FUNCTION MeasureUnits_to_Count : int;
VAR_INPUT
	iValue_in	: INT; 
	iHigh		: REAL;
	iLow		: REAL;
END_VAR
VAR
END_VAR

MeasureUnits_to_Count	:=	TO_INT((INT_TO_REAL(iValue_In) - iLow)*(32767.0/(iHigh - iLow)));

END_FUNCTION

(* stored: Version 1.1.0.1, ProductVersion 3.1.4024.12
   POU MeasureUnits_to_Count: Id {b1349917-8af6-4438-86a4-6346e1c26277}, SpecialFunc None *)
